// Mitsubishi GX Works2 project: test   PLC: Q02U

PROGRAM MAIN
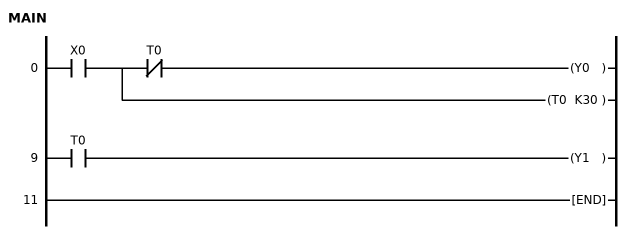
0     LD      X0
      MPS
      ANI     T0
      OUT     Y0
      MPP
      OUT     T0 K30
9     LD      T0
      OUT     Y1
11    END
END_PROGRAM
